FUNCTION_BLOCK EM_Template EXTENDS FB_EM_Base IMPLEMENTS ITF_EM_Template
VAR
// Local variables
	
// Config Struct
	s_stConfig						: ST_EM_Template_Config;
	
// Control modules
	// n.a.
	
// Inputs
	// n.a.
	
// Outputs
	// n.a.
	
// Alarms
	// n.a.
	
END_VAR

SUPER^();

METHOD PROTECTED _m_Alarms
SUPER^._m_Alarms();

// Alarm description
	// Configuration
	// n.a.
	// Call
	// n.a.
END_METHOD

METHOD PROTECTED _m_Modules
SUPER^._m_Modules();

// Description of CM
	// n.a.
END_METHOD

{attribute 'monitoring' := 'call'}
PROPERTY p_rstConfig : REFERENCE TO ST_EM_Template_Config
GET
p_rstConfig := s_stConfig;
END_GET
END_PROPERTY

END_FUNCTION_BLOCK

(* stored: Version 1.1.0.1, ProductVersion 3.1.4024.10
   POU EM_Template: Id {4c58fcab-0c4e-44d2-958d-5966280c363d}, SpecialFunc None
   Folder Basic: Id {c388fe87-eb83-464b-87de-602fe4fe0cbf}
   Folder itfEM_Template: Id {d7508406-5702-4329-8b61-48b06afc9484}
   Folder OMAC PackML: Id {3a08366a-ef8f-4f92-b7f1-5e107f704d0d}
   Method _m_Alarms: Id {305634a4-4787-42f7-a478-02ef40ad8999}
   Method _m_Modules: Id {18e9756f-350b-4c62-ae92-97b2dd506529}
   Property p_rstConfig: Id {511eb571-1518-4b73-8dd5-92b5a3f3cd4c}
   Get Get: Id {57648b8b-7208-4205-947c-0f251eebf744} *)
